// SIMATIC S7-200 SMART project (STEP 7-Micro/WIN SMART), CPU ST40

ORGANIZATION_BLOCK MAIN:OB1
TITLE=程序注释
BEGIN
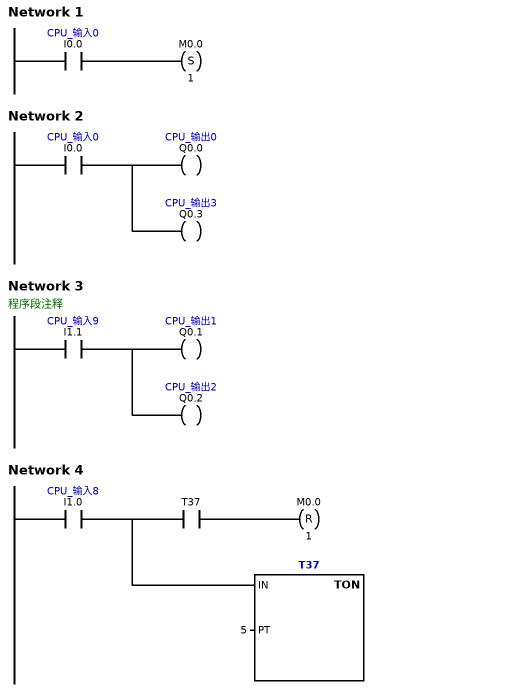
Network 1
LD     CPU_输入0:I0.0
S      M0.0, 1
Network 2
LD     CPU_输入0:I0.0
=      CPU_输出0:Q0.0
=      CPU_输出3:Q0.3
Network 3
// 程序段注释
LD     CPU_输入9:I1.1
=      CPU_输出1:Q0.1
=      CPU_输出2:Q0.2
Network 4
LD     CPU_输入8:I1.0
LPS
A      T37
R      M0.0, 1
LPP
TON    T37, 5
END_ORGANIZATION_BLOCK
